PROGRAM P_Outputs
VAR
END_VAR

///////////////////// Lights //////////////////////////////


IF G_Buttons.bManualModeSelector OR G_Buttons.bAutoModeSelector THEN
	G_Outputs.bGreenButtonLight := FALSE;
	G_Outputs.bRedButtonLight := TRUE;
ELSE
	G_Outputs.bGreenButtonLight := TRUE;
	G_Outputs.bRedButtonLight := FALSE;
END_IF

END_PROGRAM

(* stored: Version 1.1.0.1, ProductVersion 3.1.4024.12
   POU P_Outputs: Id {05725e2c-789e-4faf-9ddc-3f7ec72a2093}, SpecialFunc None *)
